# EPICS autosave request: soft_iocs/labjack/iocBoot/ioclabjack/auto_settings.req
file "LabJack_T4_settings.req", P=$(P)
file "LabJack_T4_settings.req", P=$(P2)
file "LabJack_T4_settings.req", P=$(P3)
